FUNCTION_BLOCK MatrixCsvReader
VAR_IN_OUT CONSTANT
	M : Matrix;
END_VAR
VAR_INPUT
	bExecute : BOOL;
	sPathName : T_MaxString;
	tTimeout : TIME;//timeout applied indidivudally to each file operation
	nHeaderLines : UDINT;//number of lines to skip at the beginning
END_VAR
VAR_OUTPUT
	bBusy : BOOL;
	bError : BOOL;
	nErrId : UDINT;
	nErrStep : UDINT;
	nRows : UINT;
	nCols : UINT;
	nVals : UINT;
END_VAR
VAR
	FileOpen : FB_FileOpen;
	CsvRead : FB_CSVMemBufferReader;
	FileRead : FB_FileRead;
	FileSeek : FB_FileSeek;
	FileClose : FB_FileClose;
	
	hFile : UINT;
	readEOF : BOOL;
	bytesRead : DINT;
	bytesParsed : DINT;
	buffer : STRING(bufferSize);
	step : UDINT;
	
	Hi : UINT;
	Ri : UINT;
	Ci : UINT;
	BuffCmd : E_EnumCmdType;
END_VAR
VAR CONSTANT
	bufferSize : UDINT := 1024;
	dataSize : UDINT := 16;	

	stepReady : UDINT := 0;
	stepOpenFile : UDINT := 1;
	stepFillBuffer : UDINT := 2;
	stepReadBuffer : UDINT := 3;
	stepMovePointer : UDINT := 4;
	stepCloseFile : UDINT := 5;
	stepDone : UDINT := 6;
END_VAR

FileOpen(
	sNetId := '',
	sPathName := spathname,
	nMode := FOPEN_MODEREAD OR FOPEN_MODEBINARY,
	ePath := E_OpenPath.PATH_GENERIC,
	bExecute := step = stepOpenFile,
	tTimeout := tTimeout);
FileRead(snetId := '',
	hFile := hFile,
	pReadBuff := ADR(buffer),
	cbReadLen := bufferSize,
	bExecute := step = stepFillBuffer,
	tTimeout := tTimeout);
FileSeek(snetID := '',
	hFile := hFile,
	//nSeekPos := 0,
	eOrigin := E_SeekOrigin.SEEK_CUR,
	bExecute := step = stepMovePointer,
	tTimeout := tTimeout);
FileClose(
	snetId := '',
	hFile := hFile,
	bexecute := step = stepCloseFile,
	tTimeout := tTimeout);
			
CASE step OF
	stepReady:
		bError := FALSE;
		nErrId := 0;
		nErrStep := 0;
		
		hFile := 0;
		readEOF := FALSE;
		
		Hi := 0;
		Ri := 0;
		Ci := 0;
		nRows := 0;
		nCols := 0;
		
		IF bExecute THEN
			IF NOT M.IsEmpty THEN
				bBusy := TRUE;
				step := stepOpenFile;
			END_IF
		END_IF
		
	stepOpenFile:
		
		IF FileOpen.bError THEN
			bError := TRUE;
			nErrId := FileOpen.nErrId;
			nErrStep := step;
			step := stepDone;
		ELSIF NOT(FileOpen.bBusy) THEN
			hFile := FileOpen.hFile;
			step := stepFillBuffer;
		END_IF
		
	stepFillBuffer:
		bytesRead := 0;
		IF FileRead.bError THEN
			bError := TRUE;
			nErrId := FileRead.nErrId;
			nErrStep := step;
			step := stepCloseFile;
		ELSIF NOT(FileRead.bBusy) THEN
			bytesRead := UDINT_TO_DINT(FileRead.cbRead);
			readEOF := FileRead.bEOF;//it looks like EOF is mutually exclusive with actually reading bytes. so kind of useless.
			IF bytesRead = 0 THEN
				step := stepCloseFile;
			ELSE
				step := stepReadBuffer;
			END_IF
		END_IF
		
	stepReadBuffer:
		BuffCmd := E_EnumCmdType.eEnumCmd_First;
		bytesParsed := 0;
		REPEAT
			CsvRead(eCmd := BuffCmd,
				pBuffer := ADR(Buffer),
				cbBuffer := DINT_TO_UDINT(bytesRead));
			BuffCmd := E_EnumCmdType.eEnumCmd_Next;
			
			IF CsvRead.bOk THEN
				bytesparsed := bytesparsed + UDINT_TO_DINT(CsvRead.cbRead);
				IF Hi < nHeaderLines THEN
					IF CsvRead.bCRLF THEN
						Hi := Hi + 1;
					END_IF
				ELSE
					IF Ri >= M.Rows OR Ci >= M.Cols THEN
						bError := TRUE;
						nErrId :=1;
						nErrStep := step;
						step := stepCloseFile;
						RETURN;
					END_IF
					M.SetRC(Ri,Ci,STRING_TO_LREAL(CsvRead.getValue));
					Ci := Ci + 1;
					nVals := NVals + 1;
					IF CsvRead.bCRLF THEN
						Ri := Ri + 1;
						Ci := 0;
						nRows := Ri;
					END_IF
					IF Ci > nCols THEN
						nCols := Ci;
					END_IF
				END_IF
			END_IF
		UNTIL
			NOT(CsvRead.bOk)
		END_REPEAT
		IF readEOF THEN//this probably will never happen because EOF seems to be mutually exclusive with reading bytes
			step := stepCloseFile;
		ELSE
			//move pointer backwards to where it was before the read, then forward based on how much data was read from the CSV buffer. This re-reads any partial cells that were not parsed
			FileSeek.nSeekPos := bytesParsed - bytesRead;
			IF FileSeek.nSeekPos <> 0 THEN
				step := stepMovePointer;
			ELSE
				step := stepFillBuffer;
			END_IF;
		END_IF
		
	
		
	stepMovePointer:
		IF FileSeek.bError AND NOT bError THEN
			bError := TRUE;
			nErrId := FileSeek.nErrId;
			nErrStep := step;
			step := stepDone;
		ELSIF NOT(FileSeek.bBusy) THEN
			step := stepFillBuffer;
		END_IF
		
	stepCloseFile:
		
		IF FileClose.bError AND NOT bError THEN
			bError := TRUE;
			nErrId := FileClose.nErrId;
			nErrStep := step;
			step := stepDone;
		ELSIF NOT(FileClose.bBusy) THEN
			step := stepDone;
		END_IF
		
		
	stepDone:
		bBusy := FALSE;
END_CASE

IF NOT bExecute THEN
	step := stepReady;
	bBusy := FALSE;
END_IF

END_FUNCTION_BLOCK

(* stored: Version 1.1.0.1, ProductVersion 3.1.4024.9
   POU MatrixCsvReader: Id {57e330de-3a6c-0c50-1c55-a24f6c132b53}, SpecialFunc None *)
